# B&R Automation Studio project DivertAlignmentTool
Automation Studio 4.12.3.127 SP; technology packages: mapp 5.23.0, mappCockpit 5.23.0, mappMotion 5.23.0, mappView 5.23.0

## Configuration MaintTracker

CPU PC_any, AutomationRuntime C4.93, Build 4.1.2, Safety 0.0, Vc V4.72.8

### Task classes (Cpu.sw)
```
Cyclic#1 (cycle 1600 us):
  AssemblyCt <- SampleTrakCode.AssemblyCtrl.prg
Cyclic#4 (cycle 4000 us):
  GatherInfo <- DivertAlignment.GatherInfo.prg
DataObjects: McAcpSys
NcDataObjects: McDriveLog
Binaries: arsvcreg, udbdef, mvLoader, arflatprv, McAcpDrv, arcoal, TCData, FWRules, TCLang, TC, ashwac, User, sysconf, RecipeCfg, asfw, arconfig, ashwd, iomap, Role, ExCfg_2, ExCfg_1, ExCfg_3, ExCfg_5, ExCfg_4, Config_1, Config_4, Config_5, Config_3, Config_2, McProfGen, McAcpSim
Libraries: MultiUpStn, TrkBufLib, McBase, MpBase, MpAlarmX, astime, runtime, MpFile, FileIO, MpRecipe, sys_lib, MpUserX, MpServer, McAxis, McAcpTrak, standard, AsBrStr, AsIecCon, AsIODiag, arssl, aseth, ashw, arcert, aruser, dataobj, asusb, powerlnk, brsystem, AsARCfg, McAcpPar, DvAlnLib, CoTrace, AsZip
```

### Hardware
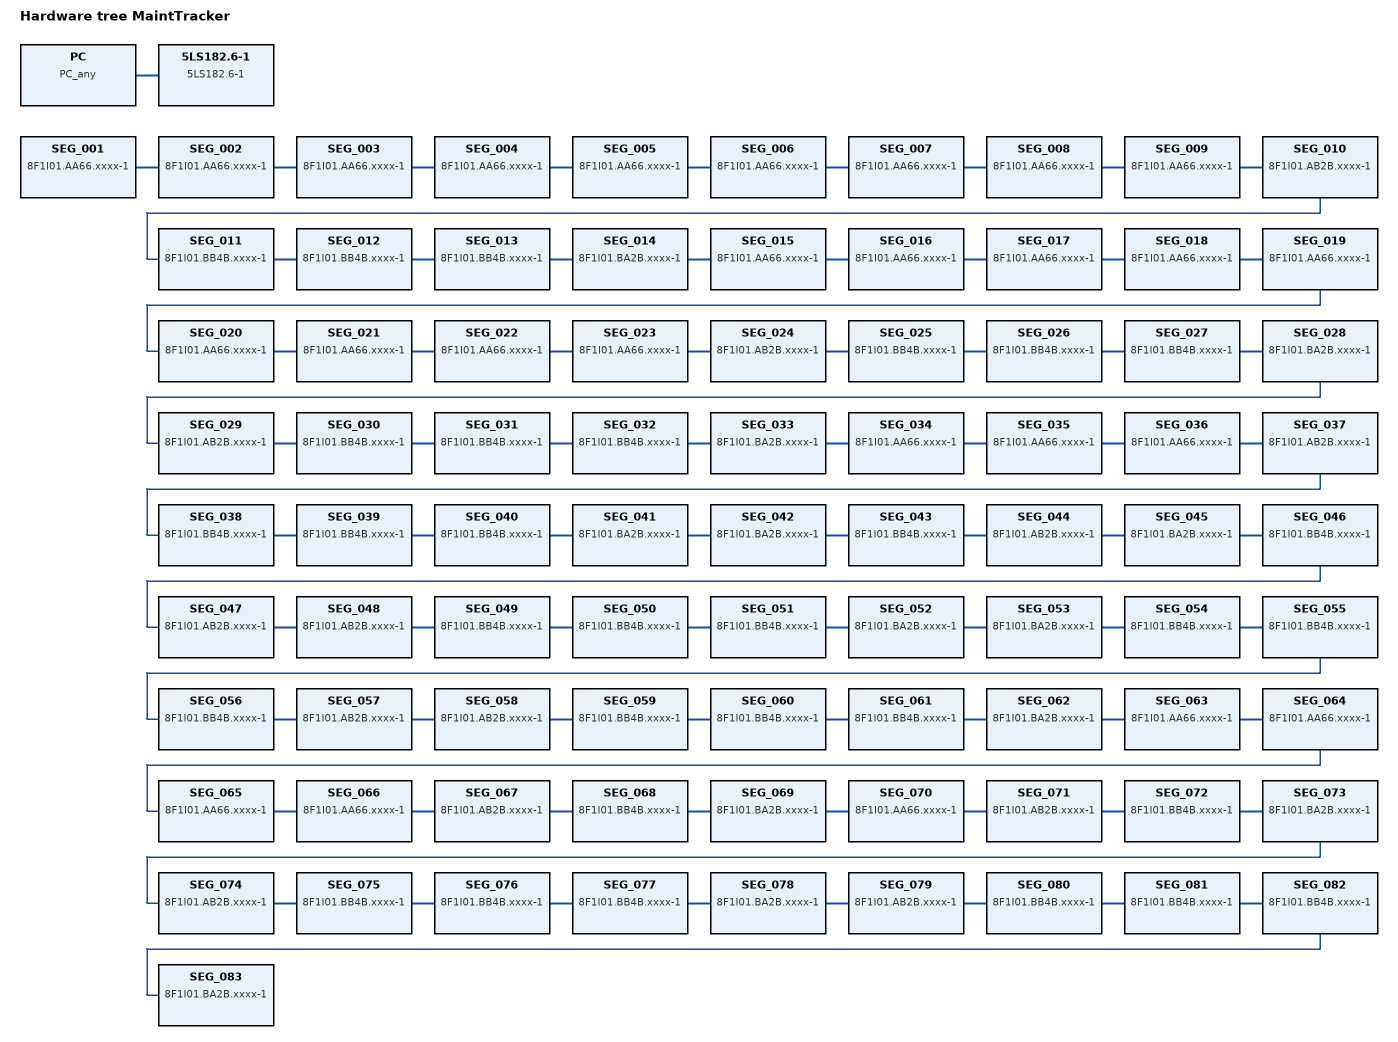
```
5LS182.6-1 : 5LS182.6-1 v1.6.0.0  [SL -> PC.SL1]
PC : PC_any v1.1.1.0 (OrderNumber=PC)
  ConfigurationID = MaintTracker_MaintTracker
  PermanentPvSize = 207088
  RemanentGlobalPvSize = 160640
  VolatileGlobalPvSize = 700000
  MotionLoggerSize = 2048000
  SystemTick = 800
  Cyclic1Duration = 1600
  Cyclic2Duration = 2400
  Cyclic2Tolerance = 10000800
  Cyclic3Duration = 3200
  Cyclic4Duration = 4000
  Cyclic5Duration = 4800
  Cyclic5Tolerance = 9984000
  Cyclic6Duration = 5600
  Cyclic6Tolerance = 12000800
  Cyclic7Duration = 6400
  Cyclic8Duration = 1600
  FileDevice1
  FileDeviceName1 = SvgData
  FileDevicePath1 = C:\projects\DivertAlignmentTool
  ActivateOpcUa = 1
  OpcUa_Limits_MonitoredItemsPerSubscription = 2000
  OpcUaInformationModels_PV_Version = 1
SEG_001 : 8F1I01.AA66.xxxx-1 v1.0.0.2  [PLK2 -> SEG_002.PLK1 [Cable Type=PowerlinkCable, Length=10, Version=1.0.0.3]; PLK3 -> 5LS182.6-1.IF1 [Cable Type=PowerlinkCable, Length=10, Version=1.0.0.3]]
  DriveConfiguration:
    McTypeID = LLMConfig
  DriveConfiguration/Segment:
    Shape = STRAIGHT660
    SegmentReference = SEG_001
    SegmentSectorDirection = Positive
    ElongationCompensation = UseAssemblySetting
    StopReaction = UseAssemblySetting
    SpeedFilter = UseAssemblySetting
    PositionControllerLagMonitor = UseAssemblySetting
SEG_002 : 8F1I01.AA66.xxxx-1 v1.0.0.2  [PLK1 -> SEG_001.PLK2 [Cable Type=PowerlinkCable, Length=10, Version=1.0.0.3]; PLK2 -> SEG_003.PLK1 [Cable Type=PowerlinkCable, Length=10, Version=1.0.0.3]]
  DriveConfiguration:
    McTypeID = LLMConfig
  DriveConfiguration/Segment:
    Shape = STRAIGHT660
    SegmentReference = SEG_002
    SegmentSectorDirection = Positive
    ElongationCompensation = UseAssemblySetting
    StopReaction = UseAssemblySetting
    SpeedFilter = UseAssemblySetting
    PositionControllerLagMonitor = UseAssemblySetting
SEG_003 : 8F1I01.AA66.xxxx-1 v1.0.0.2  [PLK1 -> SEG_002.PLK2 [Cable Type=PowerlinkCable, Length=10, Version=1.0.0.3]; PLK2 -> SEG_004.PLK1 [Cable Type=PowerlinkCable, Length=10, Version=1.0.0.3]]
  DriveConfiguration:
    McTypeID = LLMConfig
  DriveConfiguration/Segment:
    Shape = STRAIGHT660
    SegmentReference = SEG_003
    SegmentSectorDirection = Positive
    ElongationCompensation = UseAssemblySetting
    StopReaction = UseAssemblySetting
    SpeedFilter = UseAssemblySetting
    PositionControllerLagMonitor = UseAssemblySetting
SEG_004 : 8F1I01.AA66.xxxx-1 v1.0.0.2  [PLK1 -> SEG_003.PLK2 [Cable Type=PowerlinkCable, Length=10, Version=1.0.0.3]; PLK2 -> SEG_005.PLK1 [Cable Type=PowerlinkCable, Length=10, Version=1.0.0.3]]
  DriveConfiguration:
    McTypeID = LLMConfig
  DriveConfiguration/Segment:
    Shape = STRAIGHT660
    SegmentReference = SEG_004
    SegmentSectorDirection = Positive
    ElongationCompensation = UseAssemblySetting
    StopReaction = UseAssemblySetting
    SpeedFilter = UseAssemblySetting
    PositionControllerLagMonitor = UseAssemblySetting
SEG_005 : 8F1I01.AA66.xxxx-1 v1.0.0.2  [PLK1 -> SEG_004.PLK2 [Cable Type=PowerlinkCable, Length=10, Version=1.0.0.3]; PLK2 -> SEG_006.PLK1 [Cable Type=PowerlinkCable, Length=10, Version=1.0.0.3]]
  DriveConfiguration:
    McTypeID = LLMConfig
  DriveConfiguration/Segment:
    Shape = STRAIGHT660
    SegmentReference = SEG_005
    SegmentSectorDirection = Positive
    ElongationCompensation = UseAssemblySetting
    StopReaction = UseAssemblySetting
    SpeedFilter = UseAssemblySetting
    PositionControllerLagMonitor = UseAssemblySetting
SEG_006 : 8F1I01.AA66.xxxx-1 v1.0.0.2  [PLK1 -> SEG_005.PLK2 [Cable Type=PowerlinkCable, Length=10, Version=1.0.0.3]; PLK2 -> SEG_007.PLK1 [Cable Type=PowerlinkCable, Length=10, Version=1.0.0.3]]
  DriveConfiguration:
    McTypeID = LLMConfig
  DriveConfiguration/Segment:
    Shape = STRAIGHT660
    SegmentReference = SEG_006
    SegmentSectorDirection = Positive
    ElongationCompensation = UseAssemblySetting
    StopReaction = UseAssemblySetting
    SpeedFilter = UseAssemblySetting
    PositionControllerLagMonitor = UseAssemblySetting
SEG_007 : 8F1I01.AA66.xxxx-1 v1.0.0.2  [PLK1 -> SEG_006.PLK2 [Cable Type=PowerlinkCable, Length=10, Version=1.0.0.3]; PLK2 -> SEG_008.PLK1 [Cable Type=PowerlinkCable, Length=10, Version=1.0.0.3]]
  DriveConfiguration:
    McTypeID = LLMConfig
  DriveConfiguration/Segment:
    Shape = STRAIGHT660
    SegmentReference = SEG_007
    SegmentSectorDirection = Positive
    ElongationCompensation = UseAssemblySetting
    StopReaction = UseAssemblySetting
    SpeedFilter = UseAssemblySetting
    PositionControllerLagMonitor = UseAssemblySetting
SEG_008 : 8F1I01.AA66.xxxx-1 v1.0.0.2  [PLK1 -> SEG_007.PLK2 [Cable Type=PowerlinkCable, Length=10, Version=1.0.0.3]; PLK2 -> SEG_009.PLK1 [Cable Type=PowerlinkCable, Length=10, Version=1.0.0.3]]
  DriveConfiguration:
    McTypeID = LLMConfig
  DriveConfiguration/Segment:
    Shape = STRAIGHT660
    SegmentReference = SEG_008
    SegmentSectorDirection = Positive
    ElongationCompensation = UseAssemblySetting
    StopReaction = UseAssemblySetting
    SpeedFilter = UseAssemblySetting
    PositionControllerLagMonitor = UseAssemblySetting
SEG_009 : 8F1I01.AA66.xxxx-1 v1.0.0.2  [PLK1 -> SEG_008.PLK2 [Cable Type=PowerlinkCable, Length=10, Version=1.0.0.3]; PLK2 -> SEG_010.PLK1 [Cable Type=PowerlinkCable, Length=10, Version=1.0.0.3]]
  DriveConfiguration:
    McTypeID = LLMConfig
  DriveConfiguration/Segment:
    Shape = STRAIGHT660
    SegmentReference = SEG_009
    SegmentSectorDirection = Positive
    ElongationCompensation = UseAssemblySetting
    StopReaction = UseAssemblySetting
    SpeedFilter = UseAssemblySetting
    PositionControllerLagMonitor = UseAssemblySetting
SEG_010 : 8F1I01.AB2B.xxxx-1 v1.0.0.2  [PLK1 -> SEG_009.PLK2 [Cable Type=PowerlinkCable, Length=10, Version=1.0.0.3]; PLK2 -> SEG_011.PLK1 [Cable Type=PowerlinkCable, Length=10, Version=1.0.0.3]]
  DriveConfiguration:
    McTypeID = LLMConfig
  DriveConfiguration/Segment:
    Shape = STRAIGHT105_TO_CIRCULAR
    SegmentReference = SEG_010
    SegmentSectorDirection = Positive
    ElongationCompensation = UseAssemblySetting
    StopReaction = UseAssemblySetting
    SpeedFilter = UseAssemblySetting
    PositionControllerLagMonitor = UseAssemblySetting
SEG_011 : 8F1I01.BB4B.xxxx-1 v1.0.0.2  [PLK1 -> SEG_010.PLK2 [Cable Type=PowerlinkCable, Length=10, Version=1.0.0.3]; PLK2 -> SEG_012.PLK1 [Cable Type=PowerlinkCable, Length=10, Version=1.0.0.3]]
  DriveConfiguration:
    McTypeID = LLMConfig
  DriveConfiguration/Segment:
    Shape = CIRCULAR
    SegmentReference = SEG_011
    SegmentSectorDirection = Positive
    ElongationCompensation = UseAssemblySetting
    StopReaction = UseAssemblySetting
    SpeedFilter = UseAssemblySetting
    PositionControllerLagMonitor = UseAssemblySetting
SEG_012 : 8F1I01.BB4B.xxxx-1 v1.0.0.2  [PLK1 -> SEG_011.PLK2 [Cable Type=PowerlinkCable, Length=10, Version=1.0.0.3]; PLK2 -> SEG_013.PLK1 [Cable Type=PowerlinkCable, Length=10, Version=1.0.0.3]]
  DriveConfiguration:
    McTypeID = LLMConfig
  DriveConfiguration/Segment:
    Shape = CIRCULAR
    SegmentReference = SEG_012
    SegmentSectorDirection = Positive
    ElongationCompensation = UseAssemblySetting
    StopReaction = UseAssemblySetting
    SpeedFilter = UseAssemblySetting
    PositionControllerLagMonitor = UseAssemblySetting
SEG_013 : 8F1I01.BB4B.xxxx-1 v1.0.0.2  [PLK1 -> SEG_012.PLK2 [Cable Type=PowerlinkCable, Length=10, Version=1.0.0.3]; PLK2 -> SEG_014.PLK1 [Cable Type=PowerlinkCable, Length=10, Version=1.0.0.3]]
  DriveConfiguration:
    McTypeID = LLMConfig
  DriveConfiguration/Segment:
    Shape = CIRCULAR
    SegmentReference = SEG_013
    SegmentSectorDirection = Positive
    ElongationCompensation = UseAssemblySetting
    StopReaction = UseAssemblySetting
    SpeedFilter = UseAssemblySetting
    PositionControllerLagMonitor = UseAssemblySetting
SEG_014 : 8F1I01.BA2B.xxxx-1 v1.0.0.2  [PLK1 -> SEG_013.PLK2 [Cable Type=PowerlinkCable, Length=10, Version=1.0.0.3]; PLK2 -> SEG_015.PLK1 [Cable Type=PowerlinkCable, Length=10, Version=1.0.0.3]]
  DriveConfiguration:
    McTypeID = LLMConfig
  DriveConfiguration/Segment:
    Shape = CIRCULAR_TO_STRAIGHT105
    SegmentReference = SEG_014
    SegmentSectorDirection = Positive
    ElongationCompensation = UseAssemblySetting
    StopReaction = UseAssemblySetting
    SpeedFilter = UseAssemblySetting
    PositionControllerLagMonitor = UseAssemblySetting
SEG_015 : 8F1I01.AA66.xxxx-1 v1.0.0.2  [PLK1 -> SEG_014.PLK2 [Cable Type=PowerlinkCable, Length=10, Version=1.0.0.3]; PLK2 -> SEG_016.PLK1 [Cable Type=PowerlinkCable, Length=10, Version=1.0.0.3]]
  DriveConfiguration:
    McTypeID = LLMConfig
  DriveConfiguration/Segment:
    Shape = STRAIGHT660
    SegmentReference = SEG_015
    SegmentSectorDirection = Positive
    ElongationCompensation = UseAssemblySetting
    StopReaction = UseAssemblySetting
    SpeedFilter = UseAssemblySetting
    PositionControllerLagMonitor = UseAssemblySetting
SEG_016 : 8F1I01.AA66.xxxx-1 v1.0.0.2  [PLK1 -> SEG_015.PLK2 [Cable Type=PowerlinkCable, Length=10, Version=1.0.0.3]; PLK2 -> SEG_017.PLK1 [Cable Type=PowerlinkCable, Length=10, Version=1.0.0.3]]
  DriveConfiguration:
    McTypeID = LLMConfig
  DriveConfiguration/Segment:
    Shape = STRAIGHT660
    SegmentReference = SEG_016
    SegmentSectorDirection = Positive
    ElongationCompensation = UseAssemblySetting
    StopReaction = UseAssemblySetting
    SpeedFilter = UseAssemblySetting
    PositionControllerLagMonitor = UseAssemblySetting
SEG_017 : 8F1I01.AA66.xxxx-1 v1.0.0.2  [PLK1 -> SEG_016.PLK2 [Cable Type=PowerlinkCable, Length=10, Version=1.0.0.3]; PLK2 -> SEG_018.PLK1 [Cable Type=PowerlinkCable, Length=10, Version=1.0.0.3]]
  DriveConfiguration:
    McTypeID = LLMConfig
  DriveConfiguration/Segment:
    Shape = STRAIGHT660
    SegmentReference = SEG_017
    SegmentSectorDirection = Positive
    ElongationCompensation = UseAssemblySetting
    StopReaction = UseAssemblySetting
    SpeedFilter = UseAssemblySetting
    PositionControllerLagMonitor = UseAssemblySetting
SEG_018 : 8F1I01.AA66.xxxx-1 v1.0.0.2  [PLK1 -> SEG_017.PLK2 [Cable Type=PowerlinkCable, Length=10, Version=1.0.0.3]; PLK2 -> SEG_019.PLK1 [Cable Type=PowerlinkCable, Length=10, Version=1.0.0.3]]
  DriveConfiguration:
    McTypeID = LLMConfig
  DriveConfiguration/Segment:
    Shape = STRAIGHT660
    SegmentReference = SEG_018
    SegmentSectorDirection = Positive
    ElongationCompensation = UseAssemblySetting
    StopReaction = UseAssemblySetting
    SpeedFilter = UseAssemblySetting
    PositionControllerLagMonitor = UseAssemblySetting
SEG_019 : 8F1I01.AA66.xxxx-1 v1.0.0.2  [PLK1 -> SEG_018.PLK2 [Cable Type=PowerlinkCable, Length=10, Version=1.0.0.3]; PLK2 -> SEG_020.PLK1 [Cable Type=PowerlinkCable, Length=10, Version=1.0.0.3]]
  DriveConfiguration:
    McTypeID = LLMConfig
  DriveConfiguration/Segment:
    Shape = STRAIGHT660
    SegmentReference = SEG_019
    SegmentSectorDirection = Positive
    ElongationCompensation = UseAssemblySetting
    StopReaction = UseAssemblySetting
    SpeedFilter = UseAssemblySetting
    PositionControllerLagMonitor = UseAssemblySetting
SEG_020 : 8F1I01.AA66.xxxx-1 v1.0.0.2  [PLK1 -> SEG_019.PLK2 [Cable Type=PowerlinkCable, Length=10, Version=1.0.0.3]; PLK2 -> SEG_021.PLK1 [Cable Type=PowerlinkCable, Length=10, Version=1.0.0.3]]
  DriveConfiguration:
    McTypeID = LLMConfig
  DriveConfiguration/Segment:
    Shape = STRAIGHT660
    SegmentReference = SEG_020
    SegmentSectorDirection = Positive
    ElongationCompensation = UseAssemblySetting
    StopReaction = UseAssemblySetting
    SpeedFilter = UseAssemblySetting
    PositionControllerLagMonitor = UseAssemblySetting
SEG_021 : 8F1I01.AA66.xxxx-1 v1.0.0.2  [PLK1 -> SEG_020.PLK2 [Cable Type=PowerlinkCable, Length=10, Version=1.0.0.3]; PLK2 -> SEG_022.PLK1 [Cable Type=PowerlinkCable, Length=10, Version=1.0.0.3]]
  DriveConfiguration:
    McTypeID = LLMConfig
  DriveConfiguration/Segment:
    Shape = STRAIGHT660
    SegmentReference = SEG_021
    SegmentSectorDirection = Positive
    ElongationCompensation = UseAssemblySetting
    StopReaction = UseAssemblySetting
    SpeedFilter = UseAssemblySetting
    PositionControllerLagMonitor = UseAssemblySetting
SEG_022 : 8F1I01.AA66.xxxx-1 v1.0.0.2  [PLK1 -> SEG_021.PLK2 [Cable Type=PowerlinkCable, Length=10, Version=1.0.0.3]; PLK2 -> SEG_023.PLK1 [Cable Type=PowerlinkCable, Length=10, Version=1.0.0.3]]
  DriveConfiguration:
    McTypeID = LLMConfig
  DriveConfiguration/Segment:
    Shape = STRAIGHT660
    SegmentReference = SEG_022
    SegmentSectorDirection = Positive
    ElongationCompensation = UseAssemblySetting
    StopReaction = UseAssemblySetting
    SpeedFilter = UseAssemblySetting
    PositionControllerLagMonitor = UseAssemblySetting
SEG_023 : 8F1I01.AA66.xxxx-1 v1.0.0.2  [PLK1 -> SEG_022.PLK2 [Cable Type=PowerlinkCable, Length=10, Version=1.0.0.3]; PLK2 -> SEG_024.PLK1 [Cable Type=PowerlinkCable, Length=10, Version=1.0.0.3]]
  DriveConfiguration:
    McTypeID = LLMConfig
  DriveConfiguration/Segment:
    Shape = STRAIGHT660
    SegmentReference = SEG_023
    SegmentSectorDirection = Positive
    ElongationCompensation = UseAssemblySetting
    StopReaction = UseAssemblySetting
    SpeedFilter = UseAssemblySetting
    PositionControllerLagMonitor = UseAssemblySetting
SEG_024 : 8F1I01.AB2B.xxxx-1 v1.0.0.2  [PLK1 -> SEG_023.PLK2 [Cable Type=PowerlinkCable, Length=10, Version=1.0.0.3]; PLK2 -> SEG_025.PLK1 [Cable Type=PowerlinkCable, Length=10, Version=1.0.0.3]]
  DriveConfiguration:
    McTypeID = LLMConfig
  DriveConfiguration/Segment:
    Shape = STRAIGHT105_TO_CIRCULAR
    SegmentReference = SEG_024
    SegmentSectorDirection = Positive
    ElongationCompensation = UseAssemblySetting
    StopReaction = UseAssemblySetting
    SpeedFilter = UseAssemblySetting
    PositionControllerLagMonitor = UseAssemblySetting
SEG_025 : 8F1I01.BB4B.xxxx-1 v1.0.0.2  [PLK1 -> SEG_024.PLK2 [Cable Type=PowerlinkCable, Length=10, Version=1.0.0.3]; PLK2 -> SEG_026.PLK1 [Cable Type=PowerlinkCable, Length=10, Version=1.0.0.3]]
  DriveConfiguration:
    McTypeID = LLMConfig
  DriveConfiguration/Segment:
    Shape = CIRCULAR
    SegmentReference = SEG_025
    SegmentSectorDirection = Positive
    ElongationCompensation = UseAssemblySetting
    StopReaction = UseAssemblySetting
    SpeedFilter = UseAssemblySetting
    PositionControllerLagMonitor = UseAssemblySetting
SEG_026 : 8F1I01.BB4B.xxxx-1 v1.0.0.2  [PLK1 -> SEG_025.PLK2 [Cable Type=PowerlinkCable, Length=10, Version=1.0.0.3]; PLK2 -> SEG_027.PLK1 [Cable Type=PowerlinkCable, Length=10, Version=1.0.0.3]]
  DriveConfiguration:
    McTypeID = LLMConfig
  DriveConfiguration/Segment:
    Shape = CIRCULAR
    SegmentReference = SEG_026
    SegmentSectorDirection = Positive
    ElongationCompensation = UseAssemblySetting
    StopReaction = UseAssemblySetting
    SpeedFilter = UseAssemblySetting
    PositionControllerLagMonitor = UseAssemblySetting
SEG_027 : 8F1I01.BB4B.xxxx-1 v1.0.0.2  [PLK1 -> SEG_026.PLK2 [Cable Type=PowerlinkCable, Length=10, Version=1.0.0.3]; PLK2 -> SEG_028.PLK1 [Cable Type=PowerlinkCable, Length=10, Version=1.0.0.3]]
  DriveConfiguration:
    McTypeID = LLMConfig
  DriveConfiguration/Segment:
    Shape = CIRCULAR
    SegmentReference = SEG_027
    SegmentSectorDirection = Positive
    ElongationCompensation = UseAssemblySetting
    StopReaction = UseAssemblySetting
    SpeedFilter = UseAssemblySetting
    PositionControllerLagMonitor = UseAssemblySetting
SEG_028 : 8F1I01.BA2B.xxxx-1 v1.0.0.2  [PLK1 -> SEG_027.PLK2 [Cable Type=PowerlinkCable, Length=10, Version=1.0.0.3]; PLK2 -> SEG_029.PLK1 [Cable Type=PowerlinkCable, Length=10, Version=1.0.0.3]]
  DriveConfiguration:
    McTypeID = LLMConfig
  DriveConfiguration/Segment:
    Shape = CIRCULAR_TO_STRAIGHT105
    SegmentReference = SEG_028
    SegmentSectorDirection = Positive
    ElongationCompensation = UseAssemblySetting
    StopReaction = UseAssemblySetting
    SpeedFilter = UseAssemblySetting
    PositionControllerLagMonitor = UseAssemblySetting
SEG_029 : 8F1I01.AB2B.xxxx-1 v1.0.0.2  [PLK1 -> SEG_028.PLK2 [Cable Type=PowerlinkCable, Length=10, Version=1.0.0.3]; PLK2 -> SEG_030.PLK1 [Cable Type=PowerlinkCable, Length=10, Version=1.0.0.3]]
  DriveConfiguration:
    McTypeID = LLMConfig
  DriveConfiguration/Segment:
    Shape = STRAIGHT105_TO_CIRCULAR
    SegmentReference = SEG_029
    SegmentSectorDirection = Positive
    ElongationCompensation = UseAssemblySetting
    StopReaction = UseAssemblySetting
    SpeedFilter = UseAssemblySetting
    PositionControllerLagMonitor = UseAssemblySetting
SEG_030 : 8F1I01.BB4B.xxxx-1 v1.0.0.2  [PLK1 -> SEG_029.PLK2 [Cable Type=PowerlinkCable, Length=10, Version=1.0.0.3]; PLK2 -> SEG_031.PLK1 [Cable Type=PowerlinkCable, Length=10, Version=1.0.0.3]]
  DriveConfiguration:
    McTypeID = LLMConfig
  DriveConfiguration/Segment:
    Shape = CIRCULAR
    SegmentReference = SEG_030
    SegmentSectorDirection = Positive
    ElongationCompensation = UseAssemblySetting
    StopReaction = UseAssemblySetting
    SpeedFilter = UseAssemblySetting
    PositionControllerLagMonitor = UseAssemblySetting
SEG_031 : 8F1I01.BB4B.xxxx-1 v1.0.0.2  [PLK1 -> SEG_030.PLK2 [Cable Type=PowerlinkCable, Length=10, Version=1.0.0.3]; PLK2 -> SEG_032.PLK1 [Cable Type=PowerlinkCable, Length=10, Version=1.0.0.3]]
  DriveConfiguration:
    McTypeID = LLMConfig
  DriveConfiguration/Segment:
    Shape = CIRCULAR
    SegmentReference = SEG_031
    SegmentSectorDirection = Positive
    ElongationCompensation = UseAssemblySetting
    StopReaction = UseAssemblySetting
    SpeedFilter = UseAssemblySetting
    PositionControllerLagMonitor = UseAssemblySetting
SEG_032 : 8F1I01.BB4B.xxxx-1 v1.0.0.2  [PLK1 -> SEG_031.PLK2 [Cable Type=PowerlinkCable, Length=10, Version=1.0.0.3]; PLK2 -> SEG_033.PLK1 [Cable Type=PowerlinkCable, Length=10, Version=1.0.0.3]]
  DriveConfiguration:
    McTypeID = LLMConfig
  DriveConfiguration/Segment:
    Shape = CIRCULAR
    SegmentReference = SEG_032
    SegmentSectorDirection = Positive
    ElongationCompensation = UseAssemblySetting
    StopReaction = UseAssemblySetting
    SpeedFilter = UseAssemblySetting
    PositionControllerLagMonitor = UseAssemblySetting
SEG_033 : 8F1I01.BA2B.xxxx-1 v1.0.0.2  [PLK1 -> SEG_032.PLK2 [Cable Type=PowerlinkCable, Length=10, Version=1.0.0.3]; PLK2 -> SEG_034.PLK1 [Cable Type=PowerlinkCable, Length=10, Version=1.0.0.3]]
  DriveConfiguration:
    McTypeID = LLMConfig
  DriveConfiguration/Segment:
    Shape = CIRCULAR_TO_STRAIGHT105
    SegmentReference = SEG_033
    SegmentSectorDirection = Positive
    ElongationCompensation = UseAssemblySetting
    StopReaction = UseAssemblySetting
    SpeedFilter = UseAssemblySetting
    PositionControllerLagMonitor = UseAssemblySetting
SEG_034 : 8F1I01.AA66.xxxx-1 v1.0.0.2  [PLK1 -> SEG_033.PLK2 [Cable Type=PowerlinkCable, Length=10, Version=1.0.0.3]; PLK2 -> SEG_035.PLK1 [Cable Type=PowerlinkCable, Length=10, Version=1.0.0.3]]
  DriveConfiguration:
    McTypeID = LLMConfig
  DriveConfiguration/Segment:
    Shape = STRAIGHT660
    SegmentReference = SEG_034
    SegmentSectorDirection = Positive
    ElongationCompensation = UseAssemblySetting
    StopReaction = UseAssemblySetting
    SpeedFilter = UseAssemblySetting
    PositionControllerLagMonitor = UseAssemblySetting
SEG_035 : 8F1I01.AA66.xxxx-1 v1.0.0.2  [PLK1 -> SEG_034.PLK2 [Cable Type=PowerlinkCable, Length=10, Version=1.0.0.3]; PLK2 -> SEG_036.PLK1 [Cable Type=PowerlinkCable, Length=10, Version=1.0.0.3]]
  DriveConfiguration:
    McTypeID = LLMConfig
  DriveConfiguration/Segment:
    Shape = STRAIGHT660
    SegmentReference = SEG_035
    SegmentSectorDirection = Positive
    ElongationCompensation = UseAssemblySetting
    StopReaction = UseAssemblySetting
    SpeedFilter = UseAssemblySetting
    PositionControllerLagMonitor = UseAssemblySetting
SEG_036 : 8F1I01.AA66.xxxx-1 v1.0.0.2  [PLK1 -> SEG_035.PLK2 [Cable Type=PowerlinkCable, Length=10, Version=1.0.0.3]; PLK2 -> SEG_037.PLK1 [Cable Type=PowerlinkCable, Length=10, Version=1.0.0.3]]
  DriveConfiguration:
    McTypeID = LLMConfig
  DriveConfiguration/Segment:
    Shape = STRAIGHT660
    SegmentReference = SEG_036
    SegmentSectorDirection = Positive
    ElongationCompensation = UseAssemblySetting
    StopReaction = UseAssemblySetting
    SpeedFilter = UseAssemblySetting
    PositionControllerLagMonitor = UseAssemblySetting
SEG_037 : 8F1I01.AB2B.xxxx-1 v1.0.0.2  [PLK1 -> SEG_036.PLK2 [Cable Type=PowerlinkCable, Length=10, Version=1.0.0.3]; PLK2 -> SEG_038.PLK1 [Cable Type=PowerlinkCable, Length=10, Version=1.0.0.3]]
  DriveConfiguration:
    McTypeID = LLMConfig
  DriveConfiguration/Segment:
    Shape = STRAIGHT105_TO_CIRCULAR
    SegmentReference = SEG_037
    SegmentSectorDirection = Positive
    ElongationCompensation = UseAssemblySetting
    StopReaction = UseAssemblySetting
    SpeedFilter = UseAssemblySetting
    PositionControllerLagMonitor = UseAssemblySetting
SEG_038 : 8F1I01.BB4B.xxxx-1 v1.0.0.2  [PLK1 -> SEG_037.PLK2 [Cable Type=PowerlinkCable, Length=10, Version=1.0.0.3]; PLK2 -> SEG_039.PLK1 [Cable Type=PowerlinkCable, Length=10, Version=1.0.0.3]]
  DriveConfiguration:
    McTypeID = LLMConfig
  DriveConfiguration/Segment:
    Shape = CIRCULAR
    SegmentReference = SEG_038
    SegmentSectorDirection = Positive
    ElongationCompensation = UseAssemblySetting
    StopReaction = UseAssemblySetting
    SpeedFilter = UseAssemblySetting
    PositionControllerLagMonitor = UseAssemblySetting
SEG_039 : 8F1I01.BB4B.xxxx-1 v1.0.0.2  [PLK1 -> SEG_038.PLK2 [Cable Type=PowerlinkCable, Length=10, Version=1.0.0.3]; PLK2 -> SEG_040.PLK1 [Cable Type=PowerlinkCable, Length=10, Version=1.0.0.3]]
  DriveConfiguration:
    McTypeID = LLMConfig
  DriveConfiguration/Segment:
    Shape = CIRCULAR
    SegmentReference = SEG_039
    SegmentSectorDirection = Positive
    ElongationCompensation = UseAssemblySetting
    StopReaction = UseAssemblySetting
    SpeedFilter = UseAssemblySetting
    PositionControllerLagMonitor = UseAssemblySetting
SEG_040 : 8F1I01.BB4B.xxxx-1 v1.0.0.2  [PLK1 -> SEG_039.PLK2 [Cable Type=PowerlinkCable, Length=10, Version=1.0.0.3]; PLK2 -> SEG_041.PLK1 [Cable Type=PowerlinkCable, Length=10, Version=1.0.0.3]]
  DriveConfiguration:
    McTypeID = LLMConfig
  DriveConfiguration/Segment:
    Shape = CIRCULAR
    SegmentReference = SEG_040
    SegmentSectorDirection = Positive
    ElongationCompensation = UseAssemblySetting
    StopReaction = UseAssemblySetting
    SpeedFilter = UseAssemblySetting
    PositionControllerLagMonitor = UseAssemblySetting
SEG_041 : 8F1I01.BA2B.xxxx-1 v1.0.0.2  [PLK1 -> SEG_040.PLK2 [Cable Type=PowerlinkCable, Length=10, Version=1.0.0.3]; PLK2 -> SEG_042.PLK1 [Cable Type=PowerlinkCable, Length=10, Version=1.0.0.3]]
  DriveConfiguration:
    McTypeID = LLMConfig
  DriveConfiguration/Segment:
    Shape = CIRCULAR_TO_STRAIGHT105
    SegmentReference = SEG_041
    SegmentSectorDirection = Positive
    ElongationCompensation = UseAssemblySetting
    StopReaction = UseAssemblySetting
    SpeedFilter = UseAssemblySetting
    PositionControllerLagMonitor = UseAssemblySetting
SEG_042 : 8F1I01.BA2B.xxxx-1 v1.0.0.2  [PLK1 -> SEG_041.PLK2 [Cable Type=PowerlinkCable, Length=10, Version=1.0.0.3]; PLK2 -> SEG_043.PLK1 [Cable Type=PowerlinkCable, Length=10, Version=1.0.0.3]]
  DriveConfiguration:
    McTypeID = LLMConfig
  DriveConfiguration/Segment:
    Shape = CIRCULAR_TO_STRAIGHT105
    SegmentReference = SEG_042
    SegmentSectorDirection = Positive
    ElongationCompensation = UseAssemblySetting
    StopReaction = UseAssemblySetting
    SpeedFilter = UseAssemblySetting
    PositionControllerLagMonitor = UseAssemblySetting
SEG_043 : 8F1I01.BB4B.xxxx-1 v1.0.0.2  [PLK1 -> SEG_042.PLK2 [Cable Type=PowerlinkCable, Length=10, Version=1.0.0.3]; PLK2 -> SEG_044.PLK1 [Cable Type=PowerlinkCable, Length=10, Version=1.0.0.3]]
  DriveConfiguration:
    McTypeID = LLMConfig
  DriveConfiguration/Segment:
    Shape = CIRCULAR
    SegmentReference = SEG_043
    SegmentSectorDirection = Positive
    ElongationCompensation = UseAssemblySetting
    StopReaction = UseAssemblySetting
    SpeedFilter = UseAssemblySetting
    PositionControllerLagMonitor = UseAssemblySetting
SEG_044 : 8F1I01.AB2B.xxxx-1 v1.0.0.2  [PLK1 -> SEG_043.PLK2 [Cable Type=PowerlinkCable, Length=10, Version=1.0.0.3]; PLK2 -> SEG_045.PLK1 [Cable Type=PowerlinkCable, Length=10, Version=1.0.0.3]]
  DriveConfiguration:
    McTypeID = LLMConfig
  DriveConfiguration/Segment:
    Shape = STRAIGHT105_TO_CIRCULAR
    SegmentReference = SEG_044
    SegmentSectorDirection = Positive
    ElongationCompensation = UseAssemblySetting
    StopReaction = UseAssemblySetting
    SpeedFilter = UseAssemblySetting
    PositionControllerLagMonitor = UseAssemblySetting
SEG_045 : 8F1I01.BA2B.xxxx-1 v1.0.0.2  [PLK1 -> SEG_044.PLK2 [Cable Type=PowerlinkCable, Length=10, Version=1.0.0.3]; PLK2 -> SEG_046.PLK1 [Cable Type=PowerlinkCable, Length=10, Version=1.0.0.3]]
  DriveConfiguration:
    McTypeID = LLMConfig
  DriveConfiguration/Segment:
    Shape = CIRCULAR_TO_STRAIGHT105
    SegmentReference = SEG_045
    SegmentSectorDirection = Positive
    ElongationCompensation = UseAssemblySetting
    StopReaction = UseAssemblySetting
    SpeedFilter = UseAssemblySetting
    PositionControllerLagMonitor = UseAssemblySetting
SEG_046 : 8F1I01.BB4B.xxxx-1 v1.0.0.2  [PLK1 -> SEG_045.PLK2 [Cable Type=PowerlinkCable, Length=10, Version=1.0.0.3]; PLK2 -> SEG_047.PLK1 [Cable Type=PowerlinkCable, Length=10, Version=1.0.0.3]]
  DriveConfiguration:
    McTypeID = LLMConfig
  DriveConfiguration/Segment:
    Shape = CIRCULAR
    SegmentReference = SEG_046
    SegmentSectorDirection = Positive
    ElongationCompensation = UseAssemblySetting
    StopReaction = UseAssemblySetting
    SpeedFilter = UseAssemblySetting
    PositionControllerLagMonitor = UseAssemblySetting
SEG_047 : 8F1I01.AB2B.xxxx-1 v1.0.0.2  [PLK1 -> SEG_046.PLK2 [Cable Type=PowerlinkCable, Length=10, Version=1.0.0.3]; PLK2 -> SEG_048.PLK1 [Cable Type=PowerlinkCable, Length=10, Version=1.0.0.3]]
  DriveConfiguration:
    McTypeID = LLMConfig
  DriveConfiguration/Segment:
    Shape = STRAIGHT105_TO_CIRCULAR
    SegmentReference = SEG_047
    SegmentSectorDirection = Positive
    ElongationCompensation = UseAssemblySetting
    StopReaction = UseAssemblySetting
    SpeedFilter = UseAssemblySetting
    PositionControllerLagMonitor = UseAssemblySetting
SEG_048 : 8F1I01.AB2B.xxxx-1 v1.0.0.2  [PLK1 -> SEG_047.PLK2 [Cable Type=PowerlinkCable, Length=10, Version=1.0.0.3]; PLK2 -> SEG_049.PLK1 [Cable Type=PowerlinkCable, Length=10, Version=1.0.0.3]]
  DriveConfiguration:
    McTypeID = LLMConfig
  DriveConfiguration/Segment:
    Shape = STRAIGHT105_TO_CIRCULAR
    SegmentReference = SEG_048
    SegmentSectorDirection = Positive
    ElongationCompensation = UseAssemblySetting
    StopReaction = UseAssemblySetting
    SpeedFilter = UseAssemblySetting
    PositionControllerLagMonitor = UseAssemblySetting
SEG_049 : 8F1I01.BB4B.xxxx-1 v1.0.0.2  [PLK1 -> SEG_048.PLK2 [Cable Type=PowerlinkCable, Length=10, Version=1.0.0.3]; PLK2 -> SEG_050.PLK1 [Cable Type=PowerlinkCable, Length=10, Version=1.0.0.3]]
  DriveConfiguration:
    McTypeID = LLMConfig
  DriveConfiguration/Segment:
    Shape = CIRCULAR
    SegmentReference = SEG_049
    SegmentSectorDirection = Positive
    ElongationCompensation = UseAssemblySetting
    StopReaction = UseAssemblySetting
    SpeedFilter = UseAssemblySetting
    PositionControllerLagMonitor = UseAssemblySetting
SEG_050 : 8F1I01.BB4B.xxxx-1 v1.0.0.2  [PLK1 -> SEG_049.PLK2 [Cable Type=PowerlinkCable, Length=10, Version=1.0.0.3]; PLK2 -> SEG_051.PLK1 [Cable Type=PowerlinkCable, Length=10, Version=1.0.0.3]]
  DriveConfiguration:
    McTypeID = LLMConfig
  DriveConfiguration/Segment:
    Shape = CIRCULAR
    SegmentReference = SEG_050
    SegmentSectorDirection = Positive
    ElongationCompensation = UseAssemblySetting
    StopReaction = UseAssemblySetting
    SpeedFilter = UseAssemblySetting
    PositionControllerLagMonitor = UseAssemblySetting
SEG_051 : 8F1I01.BB4B.xxxx-1 v1.0.0.2  [PLK1 -> SEG_050.PLK2 [Cable Type=PowerlinkCable, Length=10, Version=1.0.0.3]; PLK2 -> SEG_052.PLK1 [Cable Type=PowerlinkCable, Length=10, Version=1.0.0.3]]
  DriveConfiguration:
    McTypeID = LLMConfig
  DriveConfiguration/Segment:
    Shape = CIRCULAR
    SegmentReference = SEG_051
    SegmentSectorDirection = Positive
    ElongationCompensation = UseAssemblySetting
    StopReaction = UseAssemblySetting
    SpeedFilter = UseAssemblySetting
    PositionControllerLagMonitor = UseAssemblySetting
SEG_052 : 8F1I01.BA2B.xxxx-1 v1.0.0.2  [PLK1 -> SEG_051.PLK2 [Cable Type=PowerlinkCable, Length=10, Version=1.0.0.3]; PLK2 -> SEG_053.PLK1 [Cable Type=PowerlinkCable, Length=10, Version=1.0.0.3]]
  DriveConfiguration:
    McTypeID = LLMConfig
  DriveConfiguration/Segment:
    Shape = CIRCULAR_TO_STRAIGHT105
    SegmentReference = SEG_052
    SegmentSectorDirection = Positive
    ElongationCompensation = UseAssemblySetting
    StopReaction = UseAssemblySetting
    SpeedFilter = UseAssemblySetting
    PositionControllerLagMonitor = UseAssemblySetting
SEG_053 : 8F1I01.BA2B.xxxx-1 v1.0.0.2  [PLK1 -> SEG_052.PLK2 [Cable Type=PowerlinkCable, Length=10, Version=1.0.0.3]; PLK2 -> SEG_054.PLK1 [Cable Type=PowerlinkCable, Length=10, Version=1.0.0.3]]
  DriveConfiguration:
    McTypeID = LLMConfig
  DriveConfiguration/Segment:
    Shape = CIRCULAR_TO_STRAIGHT105
    SegmentReference = SEG_053
    SegmentSectorDirection = Positive
    ElongationCompensation = UseAssemblySetting
    StopReaction = UseAssemblySetting
    SpeedFilter = UseAssemblySetting
    PositionControllerLagMonitor = UseAssemblySetting
SEG_054 : 8F1I01.BB4B.xxxx-1 v1.0.0.2  [PLK1 -> SEG_053.PLK2 [Cable Type=PowerlinkCable, Length=10, Version=1.0.0.3]; PLK2 -> SEG_055.PLK1 [Cable Type=PowerlinkCable, Length=10, Version=1.0.0.3]]
  DriveConfiguration:
    McTypeID = LLMConfig
  DriveConfiguration/Segment:
    Shape = CIRCULAR
    SegmentReference = SEG_054
    SegmentSectorDirection = Positive
    ElongationCompensation = UseAssemblySetting
    StopReaction = UseAssemblySetting
    SpeedFilter = UseAssemblySetting
    PositionControllerLagMonitor = UseAssemblySetting
SEG_055 : 8F1I01.BB4B.xxxx-1 v1.0.0.2  [PLK1 -> SEG_054.PLK2 [Cable Type=PowerlinkCable, Length=10, Version=1.0.0.3]; PLK2 -> SEG_056.PLK1 [Cable Type=PowerlinkCable, Length=10, Version=1.0.0.3]]
  DriveConfiguration:
    McTypeID = LLMConfig
  DriveConfiguration/Segment:
    Shape = CIRCULAR
    SegmentReference = SEG_055
    SegmentSectorDirection = Positive
    ElongationCompensation = UseAssemblySetting
    StopReaction = UseAssemblySetting
    SpeedFilter = UseAssemblySetting
    PositionControllerLagMonitor = UseAssemblySetting
SEG_056 : 8F1I01.BB4B.xxxx-1 v1.0.0.2  [PLK1 -> SEG_055.PLK2 [Cable Type=PowerlinkCable, Length=10, Version=1.0.0.3]; PLK2 -> SEG_057.PLK1 [Cable Type=PowerlinkCable, Length=10, Version=1.0.0.3]]
  DriveConfiguration:
    McTypeID = LLMConfig
  DriveConfiguration/Segment:
    Shape = CIRCULAR
    SegmentReference = SEG_056
    SegmentSectorDirection = Positive
    ElongationCompensation = UseAssemblySetting
    StopReaction = UseAssemblySetting
    SpeedFilter = UseAssemblySetting
    PositionControllerLagMonitor = UseAssemblySetting
SEG_057 : 8F1I01.AB2B.xxxx-1 v1.0.0.2  [PLK1 -> SEG_056.PLK2 [Cable Type=PowerlinkCable, Length=10, Version=1.0.0.3]; PLK2 -> SEG_058.PLK1 [Cable Type=PowerlinkCable, Length=10, Version=1.0.0.3]]
  DriveConfiguration:
    McTypeID = LLMConfig
  DriveConfiguration/Segment:
    Shape = STRAIGHT105_TO_CIRCULAR
    SegmentReference = SEG_057
    SegmentSectorDirection = Positive
    ElongationCompensation = UseAssemblySetting
    StopReaction = UseAssemblySetting
    SpeedFilter = UseAssemblySetting
    PositionControllerLagMonitor = UseAssemblySetting
SEG_058 : 8F1I01.AB2B.xxxx-1 v1.0.0.2  [PLK1 -> SEG_057.PLK2 [Cable Type=PowerlinkCable, Length=10, Version=1.0.0.3]; PLK2 -> SEG_059.PLK1 [Cable Type=PowerlinkCable, Length=10, Version=1.0.0.3]]
  DriveConfiguration:
    McTypeID = LLMConfig
  DriveConfiguration/Segment:
    Shape = STRAIGHT105_TO_CIRCULAR
    SegmentReference = SEG_058
    SegmentSectorDirection = Positive
    ElongationCompensation = UseAssemblySetting
    StopReaction = UseAssemblySetting
    SpeedFilter = UseAssemblySetting
    PositionControllerLagMonitor = UseAssemblySetting
SEG_059 : 8F1I01.BB4B.xxxx-1 v1.0.0.2  [PLK1 -> SEG_058.PLK2 [Cable Type=PowerlinkCable, Length=10, Version=1.0.0.3]; PLK2 -> SEG_060.PLK1 [Cable Type=PowerlinkCable, Length=10, Version=1.0.0.3]]
  DriveConfiguration:
    McTypeID = LLMConfig
  DriveConfiguration/Segment:
    Shape = CIRCULAR
    SegmentReference = SEG_059
    SegmentSectorDirection = Positive
    ElongationCompensation = UseAssemblySetting
    StopReaction = UseAssemblySetting
    SpeedFilter = UseAssemblySetting
    PositionControllerLagMonitor = UseAssemblySetting
SEG_060 : 8F1I01.BB4B.xxxx-1 v1.0.0.2  [PLK1 -> SEG_059.PLK2 [Cable Type=PowerlinkCable, Length=10, Version=1.0.0.3]; PLK2 -> SEG_061.PLK1 [Cable Type=PowerlinkCable, Length=10, Version=1.0.0.3]]
  DriveConfiguration:
    McTypeID = LLMConfig
  DriveConfiguration/Segment:
    Shape = CIRCULAR
    SegmentReference = SEG_060
    SegmentSectorDirection = Positive
    ElongationCompensation = UseAssemblySetting
    StopReaction = UseAssemblySetting
    SpeedFilter = UseAssemblySetting
    PositionControllerLagMonitor = UseAssemblySetting
SEG_061 : 8F1I01.BB4B.xxxx-1 v1.0.0.2  [PLK1 -> SEG_060.PLK2 [Cable Type=PowerlinkCable, Length=10, Version=1.0.0.3]; PLK2 -> SEG_062.PLK1 [Cable Type=PowerlinkCable, Length=10, Version=1.0.0.3]]
  DriveConfiguration:
    McTypeID = LLMConfig
  DriveConfiguration/Segment:
    Shape = CIRCULAR
    SegmentReference = SEG_061
    SegmentSectorDirection = Positive
    ElongationCompensation = UseAssemblySetting
    StopReaction = UseAssemblySetting
    SpeedFilter = UseAssemblySetting
    PositionControllerLagMonitor = UseAssemblySetting
SEG_062 : 8F1I01.BA2B.xxxx-1 v1.0.0.2  [PLK1 -> SEG_061.PLK2 [Cable Type=PowerlinkCable, Length=10, Version=1.0.0.3]; PLK2 -> SEG_063.PLK1 [Cable Type=PowerlinkCable, Length=10, Version=1.0.0.3]]
  DriveConfiguration:
    McTypeID = LLMConfig
  DriveConfiguration/Segment:
    Shape = CIRCULAR_TO_STRAIGHT105
    SegmentReference = SEG_062
    SegmentSectorDirection = Positive
    ElongationCompensation = UseAssemblySetting
    StopReaction = UseAssemblySetting
    SpeedFilter = UseAssemblySetting
    PositionControllerLagMonitor = UseAssemblySetting
SEG_063 : 8F1I01.AA66.xxxx-1 v1.0.0.2  [PLK1 -> SEG_062.PLK2 [Cable Type=PowerlinkCable, Length=10, Version=1.0.0.3]; PLK2 -> SEG_064.PLK1 [Cable Type=PowerlinkCable, Length=10, Version=1.0.0.3]]
  DriveConfiguration:
    McTypeID = LLMConfig
  DriveConfiguration/Segment:
    Shape = STRAIGHT660
    SegmentReference = SEG_063
    SegmentSectorDirection = Positive
    ElongationCompensation = UseAssemblySetting
    StopReaction = UseAssemblySetting
    SpeedFilter = UseAssemblySetting
    PositionControllerLagMonitor = UseAssemblySetting
SEG_064 : 8F1I01.AA66.xxxx-1 v1.0.0.2  [PLK1 -> SEG_063.PLK2 [Cable Type=PowerlinkCable, Length=10, Version=1.0.0.3]; PLK2 -> SEG_065.PLK1 [Cable Type=PowerlinkCable, Length=10, Version=1.0.0.3]]
  DriveConfiguration:
    McTypeID = LLMConfig
  DriveConfiguration/Segment:
    Shape = STRAIGHT660
    SegmentReference = SEG_064
    SegmentSectorDirection = Positive
    ElongationCompensation = UseAssemblySetting
    StopReaction = UseAssemblySetting
    SpeedFilter = UseAssemblySetting
    PositionControllerLagMonitor = UseAssemblySetting
SEG_065 : 8F1I01.AA66.xxxx-1 v1.0.0.2  [PLK1 -> SEG_064.PLK2 [Cable Type=PowerlinkCable, Length=10, Version=1.0.0.3]; PLK2 -> SEG_066.PLK1 [Cable Type=PowerlinkCable, Length=10, Version=1.0.0.3]]
  DriveConfiguration:
    McTypeID = LLMConfig
  DriveConfiguration/Segment:
    Shape = STRAIGHT660
    SegmentReference = SEG_065
    SegmentSectorDirection = Positive
    ElongationCompensation = UseAssemblySetting
    StopReaction = UseAssemblySetting
    SpeedFilter = UseAssemblySetting
    PositionControllerLagMonitor = UseAssemblySetting
SEG_066 : 8F1I01.AA66.xxxx-1 v1.0.0.2  [PLK1 -> SEG_065.PLK2 [Cable Type=PowerlinkCable, Length=10, Version=1.0.0.3]; PLK2 -> SEG_067.PLK1 [Cable Type=PowerlinkCable, Length=10, Version=1.0.0.3]]
  DriveConfiguration:
    McTypeID = LLMConfig
  DriveConfiguration/Segment:
    Shape = STRAIGHT660
    SegmentReference = SEG_066
    SegmentSectorDirection = Positive
    ElongationCompensation = UseAssemblySetting
    StopReaction = UseAssemblySetting
    SpeedFilter = UseAssemblySetting
    PositionControllerLagMonitor = UseAssemblySetting
SEG_067 : 8F1I01.AB2B.xxxx-1 v1.0.0.2  [PLK1 -> SEG_066.PLK2 [Cable Type=PowerlinkCable, Length=10, Version=1.0.0.3]; PLK2 -> SEG_068.PLK1 [Cable Type=PowerlinkCable, Length=10, Version=1.0.0.3]]
  DriveConfiguration:
    McTypeID = LLMConfig
  DriveConfiguration/Segment:
    Shape = STRAIGHT105_TO_CIRCULAR
    SegmentReference = SEG_067
    SegmentSectorDirection = Positive
    ElongationCompensation = UseAssemblySetting
    StopReaction = UseAssemblySetting
    SpeedFilter = UseAssemblySetting
    PositionControllerLagMonitor = UseAssemblySetting
SEG_068 : 8F1I01.BB4B.xxxx-1 v1.0.0.2  [PLK1 -> SEG_067.PLK2 [Cable Type=PowerlinkCable, Length=10, Version=1.0.0.3]; PLK2 -> SEG_069.PLK1 [Cable Type=PowerlinkCable, Length=10, Version=1.0.0.3]]
  DriveConfiguration:
    McTypeID = LLMConfig
  DriveConfiguration/Segment:
    Shape = CIRCULAR
    SegmentReference = SEG_068
    SegmentSectorDirection = Positive
    ElongationCompensation = UseAssemblySetting
    StopReaction = UseAssemblySetting
    SpeedFilter = UseAssemblySetting
    PositionControllerLagMonitor = UseAssemblySetting
SEG_069 : 8F1I01.BA2B.xxxx-1 v1.0.0.2  [PLK1 -> SEG_068.PLK2 [Cable Type=PowerlinkCable, Length=10, Version=1.0.0.3]; PLK2 -> SEG_070.PLK1 [Cable Type=PowerlinkCable, Length=10, Version=1.0.0.3]]
  DriveConfiguration:
    McTypeID = LLMConfig
  DriveConfiguration/Segment:
    Shape = CIRCULAR_TO_STRAIGHT105
    SegmentReference = SEG_069
    SegmentSectorDirection = Positive
    ElongationCompensation = UseAssemblySetting
    StopReaction = UseAssemblySetting
    SpeedFilter = UseAssemblySetting
    PositionControllerLagMonitor = UseAssemblySetting
SEG_070 : 8F1I01.AA66.xxxx-1 v1.0.0.2  [PLK1 -> SEG_069.PLK2 [Cable Type=PowerlinkCable, Length=10, Version=1.0.0.3]; PLK2 -> SEG_071.PLK1 [Cable Type=PowerlinkCable, Length=10, Version=1.0.0.3]]
  DriveConfiguration:
    McTypeID = LLMConfig
  DriveConfiguration/Segment:
    Shape = STRAIGHT660
    SegmentReference = SEG_070
    SegmentSectorDirection = Positive
    ElongationCompensation = UseAssemblySetting
    StopReaction = UseAssemblySetting
    SpeedFilter = UseAssemblySetting
    PositionControllerLagMonitor = UseAssemblySetting
SEG_071 : 8F1I01.AB2B.xxxx-1 v1.0.0.2  [PLK1 -> SEG_070.PLK2 [Cable Type=PowerlinkCable, Length=10, Version=1.0.0.3]; PLK2 -> SEG_072.PLK1 [Cable Type=PowerlinkCable, Length=10, Version=1.0.0.3]]
  DriveConfiguration:
    McTypeID = LLMConfig
  DriveConfiguration/Segment:
    Shape = STRAIGHT105_TO_CIRCULAR
    SegmentReference = SEG_071
    SegmentSectorDirection = Positive
    ElongationCompensation = UseAssemblySetting
    StopReaction = UseAssemblySetting
    SpeedFilter = UseAssemblySetting
    PositionControllerLagMonitor = UseAssemblySetting
SEG_072 : 8F1I01.BB4B.xxxx-1 v1.0.0.2  [PLK1 -> SEG_071.PLK2 [Cable Type=PowerlinkCable, Length=10, Version=1.0.0.3]; PLK2 -> SEG_073.PLK1 [Cable Type=PowerlinkCable, Length=10, Version=1.0.0.3]]
  DriveConfiguration:
    McTypeID = LLMConfig
  DriveConfiguration/Segment:
    Shape = CIRCULAR
    SegmentReference = SEG_072
    SegmentSectorDirection = Positive
    ElongationCompensation = UseAssemblySetting
    StopReaction = UseAssemblySetting
    SpeedFilter = UseAssemblySetting
    PositionControllerLagMonitor = UseAssemblySetting
SEG_073 : 8F1I01.BA2B.xxxx-1 v1.0.0.2  [PLK1 -> SEG_072.PLK2 [Cable Type=PowerlinkCable, Length=10, Version=1.0.0.3]; PLK2 -> SEG_074.PLK1 [Cable Type=PowerlinkCable, Length=10, Version=1.0.0.3]]
  DriveConfiguration:
    McTypeID = LLMConfig
  DriveConfiguration/Segment:
    Shape = CIRCULAR_TO_STRAIGHT105
    SegmentReference = SEG_073
    SegmentSectorDirection = Positive
    ElongationCompensation = UseAssemblySetting
    StopReaction = UseAssemblySetting
    SpeedFilter = UseAssemblySetting
    PositionControllerLagMonitor = UseAssemblySetting
SEG_074 : 8F1I01.AB2B.xxxx-1 v1.0.0.2  [PLK1 -> SEG_073.PLK2 [Cable Type=PowerlinkCable, Length=10, Version=1.0.0.3]; PLK2 -> SEG_075.PLK1 [Cable Type=PowerlinkCable, Length=10, Version=1.0.0.3]]
  DriveConfiguration:
    McTypeID = LLMConfig
  DriveConfiguration/Segment:
    Shape = STRAIGHT105_TO_CIRCULAR
    SegmentReference = SEG_074
    SegmentSectorDirection = Positive
    ElongationCompensation = UseAssemblySetting
    StopReaction = UseAssemblySetting
    SpeedFilter = UseAssemblySetting
    PositionControllerLagMonitor = UseAssemblySetting
SEG_075 : 8F1I01.BB4B.xxxx-1 v1.0.0.2  [PLK1 -> SEG_074.PLK2 [Cable Type=PowerlinkCable, Length=10, Version=1.0.0.3]; PLK2 -> SEG_076.PLK1 [Cable Type=PowerlinkCable, Length=10, Version=1.0.0.3]]
  DriveConfiguration:
    McTypeID = LLMConfig
  DriveConfiguration/Segment:
    Shape = CIRCULAR
    SegmentReference = SEG_075
    SegmentSectorDirection = Positive
    ElongationCompensation = UseAssemblySetting
    StopReaction = UseAssemblySetting
    SpeedFilter = UseAssemblySetting
    PositionControllerLagMonitor = UseAssemblySetting
SEG_076 : 8F1I01.BB4B.xxxx-1 v1.0.0.2  [PLK1 -> SEG_075.PLK2 [Cable Type=PowerlinkCable, Length=10, Version=1.0.0.3]; PLK2 -> SEG_077.PLK1 [Cable Type=PowerlinkCable, Length=10, Version=1.0.0.3]]
  DriveConfiguration:
    McTypeID = LLMConfig
  DriveConfiguration/Segment:
    Shape = CIRCULAR
    SegmentReference = SEG_076
    SegmentSectorDirection = Positive
    ElongationCompensation = UseAssemblySetting
    StopReaction = UseAssemblySetting
    SpeedFilter = UseAssemblySetting
    PositionControllerLagMonitor = UseAssemblySetting
SEG_077 : 8F1I01.BB4B.xxxx-1 v1.0.0.2  [PLK1 -> SEG_076.PLK2 [Cable Type=PowerlinkCable, Length=10, Version=1.0.0.3]; PLK2 -> SEG_078.PLK1 [Cable Type=PowerlinkCable, Length=10, Version=1.0.0.3]]
  DriveConfiguration:
    McTypeID = LLMConfig
  DriveConfiguration/Segment:
    Shape = CIRCULAR
    SegmentReference = SEG_077
    SegmentSectorDirection = Positive
    ElongationCompensation = UseAssemblySetting
    StopReaction = UseAssemblySetting
    SpeedFilter = UseAssemblySetting
    PositionControllerLagMonitor = UseAssemblySetting
SEG_078 : 8F1I01.BA2B.xxxx-1 v1.0.0.2  [PLK1 -> SEG_077.PLK2 [Cable Type=PowerlinkCable, Length=10, Version=1.0.0.3]; PLK2 -> SEG_079.PLK1 [Cable Type=PowerlinkCable, Length=10, Version=1.0.0.3]]
  DriveConfiguration:
    McTypeID = LLMConfig
  DriveConfiguration/Segment:
    Shape = CIRCULAR_TO_STRAIGHT105
    SegmentReference = SEG_078
    SegmentSectorDirection = Positive
    ElongationCompensation = UseAssemblySetting
    StopReaction = UseAssemblySetting
    SpeedFilter = UseAssemblySetting
    PositionControllerLagMonitor = UseAssemblySetting
SEG_079 : 8F1I01.AB2B.xxxx-1 v1.0.0.2  [PLK1 -> SEG_078.PLK2 [Cable Type=PowerlinkCable, Length=10, Version=1.0.0.3]; PLK2 -> SEG_080.PLK1 [Cable Type=PowerlinkCable, Length=10, Version=1.0.0.3]]
  DriveConfiguration:
    McTypeID = LLMConfig
  DriveConfiguration/Segment:
    Shape = STRAIGHT105_TO_CIRCULAR
    SegmentReference = SEG_079
    SegmentSectorDirection = Positive
    ElongationCompensation = UseAssemblySetting
    StopReaction = UseAssemblySetting
    SpeedFilter = UseAssemblySetting
    PositionControllerLagMonitor = UseAssemblySetting
SEG_080 : 8F1I01.BB4B.xxxx-1 v1.0.0.2  [PLK1 -> SEG_079.PLK2 [Cable Type=PowerlinkCable, Length=10, Version=1.0.0.3]; PLK2 -> SEG_081.PLK1 [Cable Type=PowerlinkCable, Length=10, Version=1.0.0.3]]
  DriveConfiguration:
    McTypeID = LLMConfig
  DriveConfiguration/Segment:
    Shape = CIRCULAR
    SegmentReference = SEG_080
    SegmentSectorDirection = Positive
    ElongationCompensation = UseAssemblySetting
    StopReaction = UseAssemblySetting
    SpeedFilter = UseAssemblySetting
    PositionControllerLagMonitor = UseAssemblySetting
SEG_081 : 8F1I01.BB4B.xxxx-1 v1.0.0.2  [PLK1 -> SEG_080.PLK2 [Cable Type=PowerlinkCable, Length=10, Version=1.0.0.3]; PLK2 -> SEG_082.PLK1 [Cable Type=PowerlinkCable, Length=10, Version=1.0.0.3]]
  DriveConfiguration:
    McTypeID = LLMConfig
  DriveConfiguration/Segment:
    Shape = CIRCULAR
    SegmentReference = SEG_081
    SegmentSectorDirection = Positive
    ElongationCompensation = UseAssemblySetting
    StopReaction = UseAssemblySetting
    SpeedFilter = UseAssemblySetting
    PositionControllerLagMonitor = UseAssemblySetting
SEG_082 : 8F1I01.BB4B.xxxx-1 v1.0.0.2  [PLK1 -> SEG_081.PLK2 [Cable Type=PowerlinkCable, Length=10, Version=1.0.0.3]; PLK2 -> SEG_083.PLK1 [Cable Type=PowerlinkCable, Length=10, Version=1.0.0.3]]
  DriveConfiguration:
    McTypeID = LLMConfig
  DriveConfiguration/Segment:
    Shape = CIRCULAR
    SegmentReference = SEG_082
    SegmentSectorDirection = Positive
    ElongationCompensation = UseAssemblySetting
    StopReaction = UseAssemblySetting
    SpeedFilter = UseAssemblySetting
    PositionControllerLagMonitor = UseAssemblySetting
SEG_083 : 8F1I01.BA2B.xxxx-1 v1.0.0.2  [PLK1 -> SEG_082.PLK2 [Cable Type=PowerlinkCable, Length=10, Version=1.0.0.3]]
  DriveConfiguration:
    McTypeID = LLMConfig
  DriveConfiguration/Segment:
    Shape = CIRCULAR_TO_STRAIGHT105
    SegmentReference = SEG_083
    SegmentSectorDirection = Positive
    ElongationCompensation = UseAssemblySetting
    StopReaction = UseAssemblySetting
    SpeedFilter = UseAssemblySetting
    PositionControllerLagMonitor = UseAssemblySetting
```

### ExCfg_1.assembly - PC/mappMotion/ExCfg_1.assembly
```
Element gAssembly_1 (Type=assembly)
  Tracks:
    TrackSeparation = 0.030
    Track[1]:
      Segments:
        SegmentRef[1] = ::SEG_001
        SegmentRef[2] = ::SEG_002
        SegmentRef[3] = ::SEG_003
        SegmentRef[4] = ::SEG_004
        SegmentRef[5] = ::SEG_005
        SegmentRef[6] = ::SEG_006
        SegmentRef[7] = ::SEG_007
        SegmentRef[8] = ::SEG_008
        SegmentRef[9] = ::SEG_009
        SegmentRef[10] = ::SEG_010
        SegmentRef[11] = ::SEG_011
        SegmentRef[12] = ::SEG_012
        SegmentRef[13] = ::SEG_013
        SegmentRef[14] = ::SEG_014
        SegmentRef[15] = ::SEG_015
        SegmentRef[16] = ::SEG_016
        SegmentRef[17] = ::SEG_017
        SegmentRef[18] = ::SEG_018
        SegmentRef[19] = ::SEG_019
        SegmentRef[20] = ::SEG_020
        SegmentRef[21] = ::SEG_021
        SegmentRef[22] = ::SEG_022
        SegmentRef[23] = ::SEG_023
        SegmentRef[24] = ::SEG_024
        SegmentRef[25] = ::SEG_025
        SegmentRef[26] = ::SEG_026
        SegmentRef[27] = ::SEG_027
        SegmentRef[28] = ::SEG_028
      Position = Absolute
        SegmentRef = ::SEG_001
        SegmentCountDirection = RightToLeft
        Translation:
          X = 0.0
          Y = 0.0
          Z = 0.0
        Orientation:
          Angle1 = 0.0
          Angle2 = 0.0
          Angle3 = 180
    Track[2]:
      Segments:
        SegmentRef[1] = ::SEG_029
        SegmentRef[2] = ::SEG_030
        SegmentRef[3] = ::SEG_031
        SegmentRef[4] = ::SEG_032
        SegmentRef[5] = ::SEG_033
        SegmentRef[6] = ::SEG_034
      Position = RelativeToOne
        TrackSegmentPosition:
          SegmentRef = ::SEG_029
        Base:
          SegmentRef = ::SEG_028
          PositionRelativeTo = FromEnd
    Track[3]:
      Segments:
        SegmentRef[1] = ::SEG_035
      Position = RelativeToOne
        TrackSegmentPosition:
          SegmentRef = ::SEG_035
          PositionRelativeTo = FromEnd
        Base:
          SegmentRef = ::SEG_034
          Position = 0.180
          PositionRelativeTo = FromEnd
    Track[4]:
      Segments:
        SegmentRef[1] = ::SEG_036
        SegmentRef[2] = ::SEG_037
        SegmentRef[3] = ::SEG_038
        SegmentRef[4] = ::SEG_039
        SegmentRef[5] = ::SEG_040
        SegmentRef[6] = ::SEG_041
      Position = RelativeToOne
        TrackSegmentPosition:
          SegmentRef = ::SEG_036
        Base:
          SegmentRef = ::SEG_035
          Position = 0.120
    Track[5]:
      Segments:
        SegmentRef[1] = ::SEG_044
        SegmentRef[2] = ::SEG_043
        SegmentRef[3] = ::SEG_042
      Position = RelativeToOne
        TrackSegmentPosition:
          SegmentRef = ::SEG_042
          PositionRelativeTo = FromEnd
        Base:
          SegmentRef = ::SEG_006
    Track[6]:
      Segments:
        SegmentRef[1] = ::SEG_047
        SegmentRef[2] = ::SEG_046
        SegmentRef[3] = ::SEG_045
      Position = RelativeToOne
        TrackSegmentPosition:
          SegmentRef = ::SEG_045
          PositionRelativeTo = FromEnd
        Base:
          SegmentRef = ::SEG_044
    Track[7]:
      Segments:
        SegmentRef[1] = ::SEG_048
        SegmentRef[2] = ::SEG_049
        SegmentRef[3] = ::SEG_050
        SegmentRef[4] = ::SEG_051
        SegmentRef[5] = ::SEG_052
      Position = RelativeToOne
        TrackSegmentPosition:
          SegmentRef = ::SEG_048
        Base:
          SegmentRef = ::SEG_016
          Position = 0.150
          PositionRelativeTo = FromEnd
    Track[8]:
      Segments:
        SegmentRef[1] = ::SEG_057
        SegmentRef[2] = ::SEG_056
        SegmentRef[3] = ::SEG_055
        SegmentRef[4] = ::SEG_054
        SegmentRef[5] = ::SEG_053
      Position = RelativeToOne
        TrackSegmentPosition:
          SegmentRef = ::SEG_053
          Position = 0
          PositionRelativeTo = FromEnd
        Base:
          SegmentRef = ::SEG_052
          Position = 0.090
          PositionRelativeTo = FromEnd
    Track[9]:
      Segments:
        SegmentRef[1] = ::SEG_058
        SegmentRef[2] = ::SEG_059
        SegmentRef[3] = ::SEG_060
        SegmentRef[4] = ::SEG_061
        SegmentRef[5] = ::SEG_062
        SegmentRef[6] = ::SEG_063
      Position = RelativeToOne
        TrackSegmentPosition:
          SegmentRef = ::SEG_058
          Position = 0
        Base:
          SegmentRef = ::SEG_057
          Position = 0.090
    Track[10]:
      Segments:
        SegmentRef[1] = ::SEG_065
        SegmentRef[2] = ::SEG_064
      Position = RelativeToOne
        TrackSegmentPosition:
          SegmentRef = ::SEG_064
          PositionRelativeTo = FromEnd
        Base:
          SegmentRef = ::SEG_063
          Position = 0.450
    Track[11]:
      Segments:
        SegmentRef[1] = ::SEG_066
        SegmentRef[2] = ::SEG_067
        SegmentRef[3] = ::SEG_068
        SegmentRef[4] = ::SEG_069
        SegmentRef[5] = ::SEG_070
        SegmentRef[6] = ::SEG_071
        SegmentRef[7] = ::SEG_072
        SegmentRef[8] = ::SEG_073
      Position = RelativeToOne
        TrackSegmentPosition:
          SegmentRef = ::SEG_066
        Base:
          SegmentRef = ::SEG_065
          Position = 0.135
    Track[12]:
      Segments:
        SegmentRef[1] = ::SEG_074
        SegmentRef[2] = ::SEG_075
        SegmentRef[3] = ::SEG_076
        SegmentRef[4] = ::SEG_077
        SegmentRef[5] = ::SEG_078
        SegmentRef[6] = ::SEG_079
        SegmentRef[7] = ::SEG_080
        SegmentRef[8] = ::SEG_081
        SegmentRef[9] = ::SEG_082
        SegmentRef[10] = ::SEG_083
      Position = RelativeToOne
        TrackSegmentPosition:
          SegmentRef = ::SEG_074
        Base:
          SegmentRef = ::SEG_022
          PositionRelativeTo = FromEnd
  CommonSegmentSettings:
    SegmentSimulationOnPLC = Off
    CoggingCompensation = Active
      UpperVelLimit = 0.5
    ElongationCompensation = Inactive
    StopReaction = InductionHalt
    SpeedFilter = NotUsed
    ControllerParameters:
      DefaultParameter:
        Controller:
          Position:
            ProportionalGain = 150
          Speed:
            ProportionalGain = 80
            IntegrationTime = 0.0
          FeedForward:
            TotalMass = 0.7
            ForcePositive = 1.5
            ForceNegative = 1.5
            SpeedForceFactor = 1.4
            ForceLoad = 0.0
        MovementErrorLimits:
          PositionError = 0.004
          VelocityError = 1.2
        Diverter:
          ForceOverride = 1.0
      AdditionalParameterSets = NotUsed
    ScopeOfErrorReaction = Assembly
    ShuttleIdentificationTime = 0
    PositionControllerLagMonitor = Inactive
    Diverter:
      DiverterWeakEndOverrideFactor = 1.0
      DiverterStrenEndOverrideFactor = 1.0
  Shuttles:
    MaxShuttleCount = 50
    MaxShuttleCommandCount = 0
    Deceleration = 0.0
    UseConvoys = Inactive
    DistanceReserve:
      Collision = 0.002
      ErrorStop = 0.006
    ShuttleStereotypes:
      ShuttleStRef[1] = ShuttleStereotype
    MagnetPlateConfigurations:
      ShuttleType[1] = 8F1SA.100.xxxxxx-x
    CollisionAvoidance:
      Strategy = Constant
      Exclusion = NotUsed
      MaximumModelDimensions:
        Length:
          ExtentToFront = 0.03
          ExtentToBack = 0.03
        Width:
          Width = 0.06
    Coupling:
      CouplingFeature:
        EliminateShuttleToShuttleDelay = FALSE
  AssemblyFeatures:
    AssemblyFeatureRef[1] = ShuttleSpawning
  Visualization:
    MonitoringPv
    ProcessingTaskClass = 4
  Alarms = None
```

### ExCfg_2.shuttlestereotype - PC/mappMotion/ExCfg_2.shuttlestereotype
```
Element ShuttleStereotype (Type=shuttlestereotype)
  MeasurementUnit = 5067858
  MeasurementResolution = 0.00001
  MovementLimits = Internal
    VelocityIsReadOnly = 0
    Velocity:
      Velocity = 4.0
    AccelerationIsReadOnly = 0
    Acceleration:
      Acceleration = 40
    DecelerationIsReadOnly = 0
    Deceleration:
      Deceleration = 40
    UpdateMode = Immediately
  JerkFilter = Used
    JerkTime = 0.02
  UserData:
    Size = 52
  StateTransitions:
    AutomaticRecontrol = Active
```

### ExCfg_3.sector - PC/mappMotion/ExCfg_3.sector
```
Element SEC_MainLoop (Type=sector)
  Type = Composed
    StartSegment:
      SegmentRef = ::SEG_001
    IntermediateSegments:
      SegmentRef[1] = ::SEG_002
      SegmentRef[2] = ::SEG_003
      SegmentRef[3] = ::SEG_004
      SegmentRef[4] = ::SEG_005
      SegmentRef[5] = ::SEG_006
      SegmentRef[6] = ::SEG_007
      SegmentRef[7] = ::SEG_008
      SegmentRef[8] = ::SEG_009
      SegmentRef[9] = ::SEG_010
      SegmentRef[10] = ::SEG_011
      SegmentRef[11] = ::SEG_012
      SegmentRef[12] = ::SEG_013
      SegmentRef[13] = ::SEG_014
      SegmentRef[14] = ::SEG_015
      SegmentRef[15] = ::SEG_016
      SegmentRef[16] = ::SEG_017
      SegmentRef[17] = ::SEG_018
      SegmentRef[18] = ::SEG_019
      SegmentRef[19] = ::SEG_020
      SegmentRef[20] = ::SEG_021
      SegmentRef[21] = ::SEG_022
      SegmentRef[22] = ::SEG_023
      SegmentRef[23] = ::SEG_024
      SegmentRef[24] = ::SEG_025
      SegmentRef[25] = ::SEG_026
      SegmentRef[26] = ::SEG_027
    EndSegment:
      SegmentRef = ::SEG_028
      PositionRelativeTo = FromEnd
  Alarms = None
Element SEC_RedHerring_1 (Type=sector)
  Type = Composed
    StartSegment:
      SegmentRef = ::SEG_017
      Position = 0.100
      PositionRelativeTo = FromEnd
    IntermediateSegments:
      SegmentRef[1] = ::SEG_018
    EndSegment:
      SegmentRef = ::SEG_019
      Position = 0.100
      PositionRelativeTo = FromEnd
  Alarms = None
Element SEC_SecondLoop (Type=sector)
  Type = Composed
    StartSegment:
      SegmentRef = ::SEG_029
    IntermediateSegments:
      SegmentRef[1] = ::SEG_030
      SegmentRef[2] = ::SEG_031
      SegmentRef[3] = ::SEG_032
      SegmentRef[4] = ::SEG_033
      SegmentRef[5] = ::SEG_034
      SegmentRef[6] = ::SEG_035
      SegmentRef[7] = ::SEG_036
      SegmentRef[8] = ::SEG_037
      SegmentRef[9] = ::SEG_038
      SegmentRef[10] = ::SEG_039
      SegmentRef[11] = ::SEG_040
    EndSegment:
      SegmentRef = ::SEG_041
      PositionRelativeTo = FromEnd
  Alarms = None
Element SEC_VolcanoLeft (Type=sector)
  Type = Composed
    StartSegment:
      SegmentRef = ::SEG_042
      PositionRelativeTo = FromEnd
    IntermediateSegments:
      SegmentRef[1] = ::SEG_043
    EndSegment:
      SegmentRef = ::SEG_044
  Alarms = None
Element SEC_VolcanoRight (Type=sector)
  Type = Composed
    StartSegment:
      SegmentRef = ::SEG_045
      PositionRelativeTo = FromEnd
    IntermediateSegments:
      SegmentRef[1] = ::SEG_046
    EndSegment:
      SegmentRef = ::SEG_047
  Alarms = None
Element SEC_Squiggle (Type=sector)
  Type = Composed
    StartSegment:
      SegmentRef = ::SEG_050
    IntermediateSegments:
      SegmentRef[1] = ::SEG_051
      SegmentRef[2] = ::SEG_052
      SegmentRef[3] = ::SEG_053
      SegmentRef[4] = ::SEG_054
      SegmentRef[5] = ::SEG_055
      SegmentRef[6] = ::SEG_056
      SegmentRef[7] = ::SEG_057
      SegmentRef[8] = ::SEG_058
      SegmentRef[9] = ::SEG_059
    EndSegment:
      SegmentRef = ::SEG_060
      PositionRelativeTo = FromEnd
  Alarms = None
Element SEC_FlipFlop (Type=sector)
  Type = Composed
    StartSegment:
      SegmentRef = ::SEG_063
      Position = 0.330
    IntermediateSegments:
      SegmentRef[1] = ::SEG_064
      SegmentRef[2] = ::SEG_065
    EndSegment:
      SegmentRef = ::SEG_066
      Position = 0.330
  Alarms = None
Element SEC_RedHerring_2 (Type=sector)
  Type = Composed
    StartSegment:
      SegmentRef = ::SEG_069
      Position = 0.100
      PositionRelativeTo = FromEnd
    IntermediateSegments:
      SegmentRef[1] = ::SEG_070
    EndSegment:
      SegmentRef = ::SEG_071
      Position = 0.100
      PositionRelativeTo = FromEnd
  Alarms = None
Element SEC_MaintenanceLoop (Type=sector)
  Type = Composed
    StartSegment:
      SegmentRef = ::SEG_077
      Position = 0.120
    IntermediateSegments:
      SegmentRef[1] = ::SEG_078
      SegmentRef[2] = ::SEG_079
    EndSegment:
      SegmentRef = ::SEG_080
      Position = 0.120
      PositionRelativeTo = FromEnd
  Alarms = None
```

### ExCfg_4.processpointlist - PC/mappMotion/ExCfg_4.processpointlist
```
Element ProcessPointList (Type=processpointlist)
```

### ExCfg_5.assemblyfeature - PC/mappMotion/ExCfg_5.assemblyfeature
```
Element ShuttleSpawning (Type=assemblyfeature)
  Type = InitShuttleSim
    InitShuttleSim[1]:
      SectorRef = SEC_MainLoop
      Orientation = Positive
      ShuttleDefinition = ShuttleSetDefinition
        StartPosition = 0.7
        NumberOfShuttles = 1
        DistnaceBetweenShuttles = 0.06
```

## Logical view

Binary libraries used (declarations not repeated): astime, runtime, FileIO, sys_lib, standard, AsBrStr, AsIecCon, AsIODiag, AsARCfg, AsZip, McBase, McAcpPar 5.23.0, McAcpTrak 5.23.0, McAxis, MpBase, MpUserX, MpAlarmX, MpFile, MpRecipe, CoTrace, MpServer

### Global.var - Global variables
```iecst
(*Global Vars*)
VAR
	gShuttles : ARRAY[0..gNUM_SHUTTLES] OF McAxisType; (*A list of references for all shuttles currently on the trak*)
	gStartTrak : BOOL;
	gStopTrak : BOOL;
	gSpawnShuttle : BOOL;
END_VAR
(*
Constants*)
VAR CONSTANT
	gNUM_SHUTTLES : USINT := 40;
END_VAR
```

### Package Logical/Libraries - Global libraries

### Library Logical/Libraries/TrkBufLib (IEC) - Implement a buffer on a track system
Depends on: standard

### Library Logical/Libraries/MultiUpStn (IEC) - This library contains a custom FUB for running stations
Depends on: TrkBufLib

#### MultiUpStn.typ - Library data types
```iecst
(*
Substation list*)

TYPE
	SubstationList_enum :
		(
		STN_1_BUFFER,
		STN_1_1,
		STN_1_2,
		STN_1_3,
		STN_1_4,
		STN_1_5,
		STN_1_6,
		STN_2_BUFFER,
		STN_2_1,
		STN_2_2,
		STN_2_3,
		STN_2_4,
		STN_2_5,
		STN_2_6,
		STN_3_BUFFER,
		STN_3_1,
		STN_3_2,
		STN_3_3,
		STN_3_4,
		STN_3_5,
		STN_3_6,
		STN_4_BUFFER,
		STN_4_1,
		STN_4_2,
		STN_4_3,
		STN_4_4,
		STN_4_5,
		STN_4_6,
		STOP_POSITION,
		SUBSTATION_COUNT
		);
END_TYPE

(*
Userdata Structure*)

TYPE
	UserDataType : 	STRUCT
		Red : REAL; (*The red value of the shuttle color*)
		Green : REAL; (*The green value of the shuttle color*)
		Blue : REAL; (*The blue value of the shuttle color*)
		Destination : SubstationDetailsType; (*The substation that the shuttle is currently being told to go to*)
		ShuttleSerialNum : STRING[12]; (*Shuttle serial number*)
		Recovered : BOOL; (*Whether or not a station has recovered the shuttle*)
	END_STRUCT;
END_TYPE

(*
Structure for information on all substations on the assembly*)

TYPE
	SubstationDetailsType : 	STRUCT
		SubstationID : SubstationList_enum; (*The enumeric "name" of this station*)
		SectorReference : UDINT; (*The reference to substation's sector*)
		ProcessPointReference : UDINT; (*The reference to substation's process point*)
		Position : LREAL; (*Offset of the substation in meters relative to the start of its sector*)
		MoveMethod : MoveMethodEnum; (*How the shuttle should be sent to the station (Absolute or Velocity)*)
	END_STRUCT;
	MoveMethodEnum :
		(
		VELOCITY,
		ABSOLUTE
		);
END_TYPE

(*
Motion parameters for substations move commands*)

TYPE
	ShMotionParType : 	STRUCT
		Velocity : REAL; (*The velocity for all shuttles on the assembly*)
		Acceleration : REAL; (*The acceleration for all shuttles on the assembly*)
		Deceleration : REAL; (*The deceleration for all shuttles on the assembly*)
	END_STRUCT;
END_TYPE

(**)
(*Structures for station FUB*)

TYPE
	StationInternalType : 	STRUCT
		BufferState : StnBufferStateEnum; (*The state of the substation's buffer*)
		SlotsState : StnSlotsStateEnum; (*The state of the substation's slots*)
		RecoveryState : StnRecoveyrStateEnum; (*The state of the substation's recovery sequence*)
		SlotEnabled : ARRAY[0..MAX_NUM_SLOTS]OF BOOL; (*1-MAX are the slots in order from closest to the buffer to farthest *)
		FarthestSlot : USINT; (*The farthest active slot in the station*)
		ActiveIndex : USINT;
		BufferIndex : USINT;
		SlotIndex : USINT;
		RecoveryIndex : USINT;
		RecovBufferIndex : USINT;
		FubIndex : USINT;
		StationBuffer : tbAsyncShuttleBufferType;
		SlotShuttleRefs : ARRAY[0..MAX_NUM_SLOTS]OF McAxisType;
		TempSlotsFilled : USINT;
		TempUserdataWritten : USINT;
		TempShuttleReleased : USINT;
		BehindBuffer : UINT;
		ActiveSlots : USINT;
		SendAway : UINT;
		RecoveryFilledSlots : BOOL;
		Fubs : StationInternalFubsType; (*The various function blocks needed for a substation*)
	END_STRUCT;
	StationInternalFubsType : 	STRUCT
		TrgPointEnable : MC_BR_TrgPointEnable_AcpTrak; (*Fub for monitoring the process point for shuttles*)
		TrgPointGetInfo : MC_BR_TrgPointGetInfo_AcpTrak; (*Fub for getting the axis reference of shuttles passing the process point*)
		ShCopyUserData : ARRAY[0..MAX_NUM_SLOTS]OF MC_BR_ShCopyUserData_AcpTrak; (*Fub for reading and writing userdata to and from the shuttle*)
		ElasticMoveAbs : ARRAY[0..MAX_NUM_SLOTS]OF MC_BR_ElasticMoveAbs_AcpTrak;
		RoutedMoveAbs : ARRAY[0..MAX_NUM_SLOTS]OF MC_BR_RoutedMoveAbs_AcpTrak; (*Fub for enacting an absolute move on the shuttle*)
		SecGetShuttleSel : MC_BR_SecGetShuttleSel_AcpTrak;
		ShReadInfo : ARRAY[0..MAX_NUM_SLOTS]OF MC_BR_ShReadInfo_AcpTrak;
		SecStop : MC_BR_SecStop_AcpTrak;
		RecoveryTimer : TON := (PT:=T#1000ms);
		ShSwitchSector : MC_BR_ShSwitchSector_AcpTrak;
		BarrierCommand : MC_BR_BarrierCommand_AcpTrak;
		BarrierReadInfo : MC_BR_BarrierReadInfo_AcpTrak;
	END_STRUCT;
	StnBufferStateEnum :
		(
		BUF_DISABLED,
		BUF_RECOVERING,
		BUF_WAIT_FOR_SH,
		BUF_READ_SH,
		BUF_PUT_ON_SECT,
		BUF_STAGE_SH,
		BUF_CLEAR_QUEUE,
		BUF_ERROR
		);
	StnSlotsStateEnum :
		(
		SLOTS_DISABLED,
		SLOTS_RECOVERING,
		SLOTS_WAIT_FOR_QUEUE,
		SLOTS_READ_USERDATA,
		SLOTS_MOVE_TO_SLOT,
		SLOTS_CONFIRM_SLOTS_FULL,
		SLOTS_WAIT_FOR_RELEASE,
		SLOTS_RELEASE_SHUTTLES,
		SLOTS_CONFIRM_RELEASE,
		SLOTS_SEND_ON,
		SLOTS_ERROR
		);
	StnRecoveyrStateEnum :
		(
		RECOV_DISABLED,
		RECOV_FIND_ALL_1,
		RECOV_PUT_ON_SECT,
		RECOV_CONFIRM_PUT_ON_SECT,
		RECOV_SEND_REVERSE,
		RECOV_CONFIRM_REVERSE,
		RECOV_FIND_ALL_2_BUFFER,
		RECOV_FIND_ALL_2,
		RECOV_SEND_FORWARD,
		RECOV_CONFIRM_FORWARD,
		RECOV_MARK_RECOVERED,
		RECOV_CHECK_REMAINING,
		RECOV_DONE,
		RECOV_ERROR
		);
END_TYPE
```

#### MultiUpStn.var - Library constants
```iecst
VAR CONSTANT
	MAX_NUM_SLOTS : USINT := 6; (*The most slots a station can have*)
	SHUTTLE_TOOLING_WIDTH : REAL := 0.1254; (*Width of the shuttle in meters (117.4 mm + 8 mm for collision avoidance)*)
	REVERSE_MOVE_OFFSET : REAL := 0.001;
	SHUTTLE_EXTENT_TO_FRONT : LREAL := 0.0587;
	SHUTTLE_WIDTH : LREAL := 0.1302;
	NUM_PPM_SAMPLES : USINT := 20;
END_VAR
```

#### MultiUpStn.fun - Library functions and function blocks
```iecst
{REDUND_ERROR} FUNCTION_BLOCK MultiUpStn (*Buffer substations distribute shuttles to the slots when given the release command*) (*$GROUP=User,$CAT=User,$GROUPICON=User.png,$CATICON=User.png*)
	VAR_INPUT
		Enable : BOOL;
		ToolingClear : BOOL;
		MotionParameters : REFERENCE TO ShMotionParType;
		SelfDetails : ARRAY[0..MAX_NUM_SLOTS] OF SubstationDetailsType; (*Index 0 is the buffer. Indeces 1-MAX are the slots in order from closest to the buffer to farthest *)
		TargetDetails : SubstationDetailsType;
		ReleaseShuttles : BOOL;
		Recover : BOOL;
		Purge : BOOL;
		ErrorReset : BOOL;
		UserData : REFERENCE TO ARRAY[0..MAX_NUM_SLOTS] OF UserDataType; (*1-MAX are the slots in order from closest to the buffer to farthest *)
	END_VAR
	VAR_OUTPUT
		FillingSlots : BOOL;
		SlotsFilled : BOOL;
		RecoveryDone : BOOL;
		Error : BOOL;
		ErrorText : STRING[100];
	END_VAR
	VAR
		Internal : StationInternalType;
	END_VAR
END_FUNCTION_BLOCK
```
